RoboDK station: Assistive_UR5e.rdk

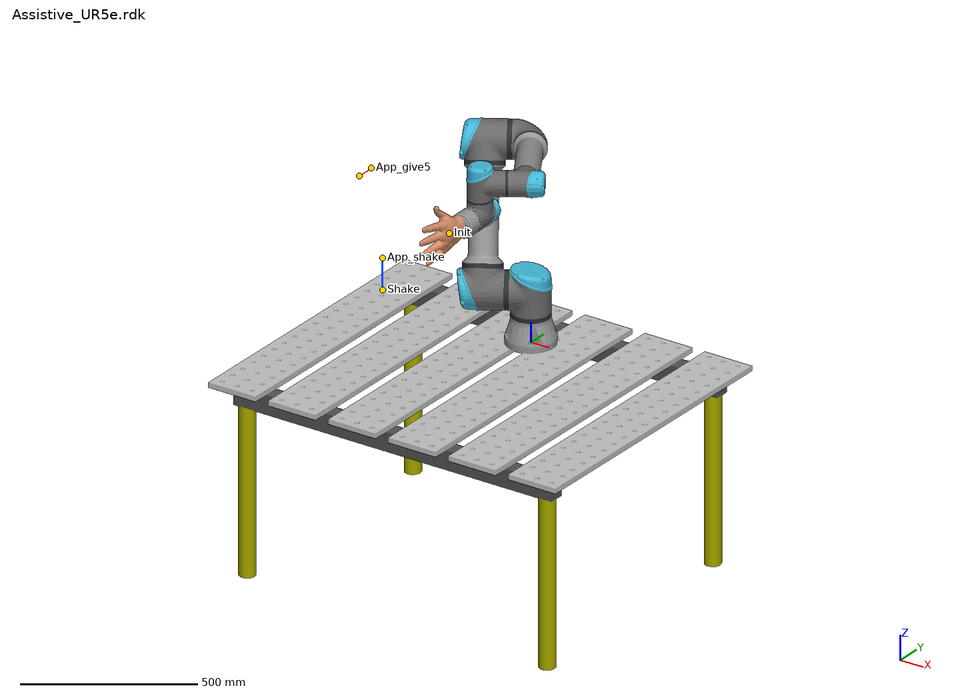
[picture v0: the station drawn from its stored meshes, robots at their saved joint values, targets as dots, program paths as lines]
Station Assistive_UR5e_SW (saved by RoboDK 5.9.2). Poses are relative to the parent item; angles as X-Y-Z fixed-axis rotations.
  - frame UR5e Base at (0, 0, 0) mm
    - robot UR5e: 6 axes, payload 5 kg, reach 850 mm, repeatability 0.03 mm, weight 18.4 kg
        modified DH rows (alpha deg, a mm, theta deg, d mm): 0, 0, 0, 162.5; 90, 0, 180, 0; 0, 425, 0, 0; 0, 392.25, 0, 133.3; -90, 0, 0, 99.7; 90, 0, 180, 99.6
        joint limits [-360, -360, -360, -360, -360, -360] to [360, 360, 360, 360, 360, 360]; home [0, -90, -90, 0, 90, 0]; saved at [-57.836, -65.392, -107.167, 172.559, -57.836, 0]
      - tool Hand, TCP at (0, 0, 50) mm, size 54.8 x 155.9 x 193.5 mm, geometry from Hand.stl
  - frame World at (0, 0, 0) mm
    - object Table at (0, 0, 0) mm, size 1193.8 x 965.2 x 609.6 mm, geometry from welding_table.sld
    - target Init (Cartesian target) at (0, -400, 500) mm, rotated rx 90 ry 0 rz 0 deg; joints [-57.836, -65.392, -107.167, 172.559, -57.836, 0] of UR5e
    - target App_shake (joint target) at (-300, -300, 300) mm, rotated rx 90 ry 0 rz 0 deg; joints [-129.97, -84.968, -123.366, -151.667, -129.97, 0] of UR5e
    - target Shake (joint target) at (-300, -300, 200) mm, rotated rx 90 ry 0 rz 0 deg; joints [-129.97, -95.332, -131.473, -133.195, -129.97, 0] of UR5e
    - target App_give5 (joint target) at (-380.86, -238.62, 533.82) mm, rotated rx 0 ry 0 rz 90 deg; joints [-130.679, -89.195, -122.013, 301.208, -90, 130.679] of UR5e
    - target Give5 (joint target) at (-380.86, -300, 533.82) mm, rotated rx 0 ry 0 rz 90 deg; joints [-125.814, -94.091, -116.939, 301.03, -90, 125.814] of UR5e
  - program Init (3 instructions, listed below)
  - program Hand_shake (5 instructions, listed below)
  - program Give_me_5! (5 instructions, listed below)
  - program MainProgram (4 instructions, listed below)
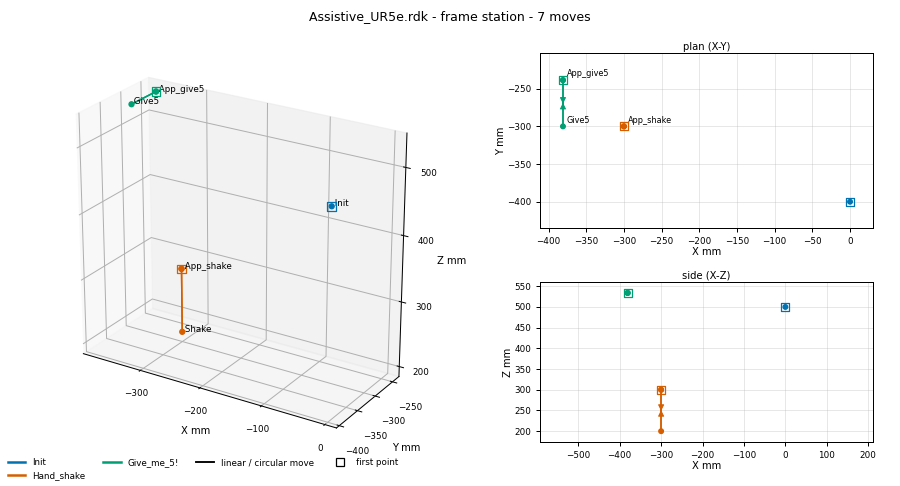
[picture p0: tool path of Assistive_UR5e.rdk in frame station, 7 of 7 moves have a stored position in this frame; points joined in program order, loops and branches not executed]

--- program Init (robot UR5e) ---
  Est. Ref.: UR5e Base
  Est. herr: Hand
  MoveJ (Init)

--- program Hand_shake (robot UR5e) ---
  Est. Ref.: UR5e Base
  Est. herr: Hand
  MoveL (App_shake)
  MoveL (Shake)
  MoveL (App_shake)

--- program Give_me_5! (robot UR5e) ---
  Est. Ref.: UR5e Base
  Est. herr: Hand
  MoveL (App_give5)
  MoveL (Give5)
  MoveL (App_give5)

--- program MainProgram (robot UR5e) ---
  Llamar Init
  Llamar Hand_shake
  Llamar Give_me_5!
  Llamar Init
